Universal Robots PolyScope program: RC_E4_Snap_440.urp

Program RC_E4_Snap_440 (createdIn=3.0.0 lastSavedIn=3.0.0 directory=/programs installation=default)
Robot Program (runOnlyOnce=true motionType=MoveJ speed=1.047198 acceleration=1.396263 useActiveTCP=false)
  'Program generated by RoboDK v4.1.0 for UR3e_HORNO on 05/09/2022 13:25:35'
  'Using nominal kinematics.'
  'Using Ref. Frame Inspeccion 02: p[-0.386000, 0.280000, -0.011500, 0.000000, 0.000000, 0.000000]'
  'Using TCP 0208-0001-0001-307-000-3 Horno: p[0.000000, 0.000000, 0.164750, 0.000000, 0.000000, 0.000000]'
  Script: set_tcp(p[0.000000, 0.000000, 0.164750, 0.000000, 0.000000, 0.000000])
  Script: movej([2.513278, -1.329928, -1.172555, -3.749812, -1.200605, 3.141595],0.60000,0.12500,0,0.0000)
  Script: movej([2.513278, -1.163858, -2.166338, -2.922100, -1.200605, 3.141595],0.60000,0.12500,0,0.0000)
  Script: movej([3.114366, -2.094744, -1.487370, -2.670179, -1.590344, 3.141593],0.60000,0.12500,0,0.0000)
  Script: movej([3.049439, -2.214125, -1.588424, -2.449744, -1.655270, 3.141593],0.60000,0.12500,0,0.0000)
  Wait Sleep waitTime=1
  Script: movej([3.310890, -2.114990, -1.770462, -2.366317, -1.393820, 3.141593],0.60000,0.12500,0,0.0000)
  Wait Sleep waitTime=1
  Script: movej([3.049439, -2.214125, -1.588424, -2.449744, -1.655270, 3.141593],0.60000,0.12500,0,0.0000)
  Wait Sleep waitTime=1
  Script: movej([2.966536, -1.779014, -2.319717, -2.153038, -1.737999, 3.141593],0.60000,0.12500,0,0.0000)
  Wait Sleep waitTime=1
  Script: movej([3.522074, -1.535541, -2.606126, -2.108009, -1.182810, 3.141593],0.60000,0.12500,0,0.0000)
  Script: movej([3.114366, -2.094744, -1.487370, -2.670179, -1.590344, 3.141593],0.60000,0.12500,0,0.0000)
  Script: movej([2.513278, -1.163858, -2.166338, -2.922100, -1.200605, 3.141595],0.60000,0.12500,0,0.0000)
  Script: movej([2.513278, -1.329928, -1.172555, -3.749812, -1.200605, 3.141595],0.60000,0.12500,0,0.0000)
